{attribute 'qualified_only'}
{attribute 'strict'}
TYPE E_Event :
(
	Verbose			:= 0,
	Debug			:= 1,
	Information		:= 2,
	Warning			:= 3,
	Error			:= 4
);
END_TYPE

(* stored: Version 1.1.0.1
   DUT E_Event: Id {d479932f-3152-0429-3151-e64105f27552} *)
